# EPICS StreamDevice protocol: echoIoc/echoApp/Db/echo.proto
write {
    out "%s";
}

read {
    in  "%s";
}

Terminator = LF;

query {
    out "\$1";
    in  "%s";
}
